{attribute addProperty BoxType "ATH2040-5250-0022"}
{attribute addProperty Id "FB_InputsAT %I*FB_Inputs_16F33527000FB_OutputsAT %Q*FB_Outputs_734938A41620WcStateAT %I*WcState_98A4DF7520.250InfoDataAT %I*InfoData_7231B2DD80100"}
{attribute addProperty CRC "1885320120"}
{attribute addProperty SizeInBites "98"}
{attribute addProperty SizeInBytes "12.25"}
TYPE ATH2040_948A301E :
STRUCT
	{attribute addProperty Name "FB_Inputs"}
	FB_Inputs : FB_Inputs_16F33527;
	{attribute addProperty Name "FB_Outputs"}
	FB_Outputs : FB_Outputs_734938A4;
	{attribute addProperty Name "WcState"}
	WcState : WcState_98A4DF75;
	{attribute addProperty Name "InfoData"}
	InfoData : InfoData_7231B2DD;
END_STRUCT
END_TYPE

(* stored: Version 1.2.0.0, ProductVersion 3.1.4024.9
   DUT ATH2040_948A301E: Id {dd832a5d-f124-4cb2-9aaa-e3e6de5613c8} *)
